FUNCTION_BLOCK FB_Light IMPLEMENTS I_LIGHT
VAR_INPUT
END_VAR
VAR_OUTPUT
END_VAR
VAR
	_rBrightness	: REAL;
	_eColor			: E_ColorCodes;
	_bIsOn			: BOOL;
END_VAR

PROPERTY bIsOn : BOOL
GET
bIsOn := _bIsOn;
END_GET
END_PROPERTY

METHOD changeBrightness : BOOL
VAR_INPUT
	in_rNewBrightness	: REAL;
END_VAR
IF in_rNewBrightness > 100.0 THEN
	_rBrightness := 100.0;
ELSIF in_rNewBrightness < 0.0 THEN
	_rBrightness := 0.0;
ELSE
	_rBrightness := in_rNewBrightness;
END_IF

ADSLOGSTR(msgCtrlMask:= ADSLOG_MSGTYPE_ERROR, msgFmtStr:= 'New Brightness: %s', strArg:= TO_STRING(_rBrightness));
END_METHOD

METHOD changeColor : BOOL
VAR_INPUT
	in_eNewColor	:E_ColorCodes;
END_VAR
_eColor := in_eNewColor;
ADSLOGSTR(msgCtrlMask:= ADSLOG_MSGTYPE_ERROR, msgFmtStr:= 'New Color: %s', strArg:= TO_STRING(_eColor));
END_METHOD

PROPERTY eColor : E_ColorCodes
GET
eColor := _eColor;
END_GET
END_PROPERTY

PROPERTY rBrightness : REAL
GET
rBrightness := _rBrightness;
END_GET
END_PROPERTY

METHOD turnLightOff : BOOL
VAR_INPUT
END_VAR
_bIsOn := FALSE;
ADSLOGSTR(msgCtrlMask:= ADSLOG_MSGTYPE_ERROR, msgFmtStr:= 'Light is off', strArg:= '');
ADSLOGSTR(msgCtrlMask:= ADSLOG_MSGTYPE_ERROR, msgFmtStr:= 'Brightness: %s', strArg:= TO_STRING(_rBrightness));
ADSLOGSTR(msgCtrlMask:= ADSLOG_MSGTYPE_ERROR, msgFmtStr:= 'Color: %s', strArg:= TO_STRING(_eColor));
END_METHOD

METHOD turnLightOn : BOOL
VAR_INPUT
END_VAR
_bIsOn := TRUE;

IF _rBrightness <= 0.0 THEN
	_rBrightness := 100.0;
END_IF

IF _eColor = E_ColorCodes.Black THEN
	_eColor := E_ColorCodes.White;
END_IF

ADSLOGSTR(msgCtrlMask:= ADSLOG_MSGTYPE_ERROR, msgFmtStr:= 'Light is on', strArg:= '');
ADSLOGSTR(msgCtrlMask:= ADSLOG_MSGTYPE_ERROR, msgFmtStr:= 'Brightness: %s', strArg:= TO_STRING(_rBrightness));
ADSLOGSTR(msgCtrlMask:= ADSLOG_MSGTYPE_ERROR, msgFmtStr:= 'Color: %s', strArg:= TO_STRING(_eColor));
END_METHOD

END_FUNCTION_BLOCK

(* stored: Version 1.1.0.1
   POU FB_Light: Id {84668e9a-79dd-49d1-a8d0-e22b0ab3419f}, SpecialFunc None
   Property bIsOn: Id {8270bcdb-2158-40e9-9bd0-190fa713dc55}
   Get Get: Id {dcbb406f-3974-452b-a5f4-ac69dcac9006}
   Method changeBrightness: Id {57f983fa-9ec0-4463-966a-c8656399e396}
   Method changeColor: Id {35832c5b-741c-468e-9d60-9df6a0411286}
   Property eColor: Id {8c3c62d0-1299-4984-a32c-b7fe4da3b262}
   Get Get: Id {75fdcde8-b065-48c1-adf8-bfd4a4cb7a49}
   Property rBrightness: Id {8300d079-f5e0-4cf7-be9a-d86a7280d1a3}
   Get Get: Id {17fc815d-3391-472d-9455-e88e81ac13af}
   Method turnLightOff: Id {cdc6f5ba-67c7-4fc7-9b0e-91eca7d205fa}
   Method turnLightOn: Id {1de21c0e-d2c3-4af7-ace3-0be53d378cc1} *)
